TYPE "InfeedWng"
VERSION : 0.1
// Block: InfeedWng
   STRUCT
      InfeedWarning : Bool;
   END_STRUCT;

END_TYPE
